TYPE IoAxisConfig EXTENDS DeviceConfiguration :
STRUCT
END_STRUCT
END_TYPE

(* stored: Version 1.1.0.1, ProductVersion 3.1.4024.12
   DUT IoAxisConfig: Id {faba0d34-7e3a-4d4c-a172-e3d03d76a500} *)
